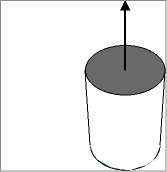
VISUALIZATION VISU_Tube_Top_6  // 167x172
VAR_IN_OUT
	azi : LREAL;
END_VAR
    Ellipse (90,120 70x50)
        p2858320360: azi
    Polygon (85,70) (165,70) (160,145) (156,155) (152,161) (146,165) (138,167) (130,170) (120,169) (111,167) (104,163) (97,159) (93,153) (90,145)
        p2858320360: azi
    Ellipse (85,45 80x50)
        p2858320360: azi
    Polygon (120,10) (125,0) (130,10)
        p2858320360: azi
    Polyline (125,70) (125,10)
        p2858320360: azi
    Polyline (160,145) (165,70)
        p2858320360: azi
    Polyline (90,145) (85,70)
        p2858320360: azi
END_VISUALIZATION

(* stored: Version 1.1.0.1, ProductVersion 3.1.4018.5
   Visu VISU_Tube_Top_6: Id {4911640f-4ada-46be-8743-85a1eccd0415} *)
